{attribute 'qualified_only'}
{attribute 'strict'}
TYPE E_AxisId :
(
	enum_member := 0,
	eAxis1		:= 1,
	eAxis2		:= 2
	
);
END_TYPE

(* stored: Version 1.1.0.1, ProductVersion 3.1.4024.4
   DUT E_AxisId: Id {e68f8c4b-466d-44e7-8668-4f676f9b4ca4} *)
